// TIA Portal V16 export
// export: Created 2021-07-12T14:47:19.1052506Z, ExportSetting WithDefaults, DisplayName Totally Integrated Automation Portal, DisplayVersion V16, DisplayName TIA Portal Version Control Interface, DisplayVersion V16, DisplayName TIA Portal Openness, DisplayVersion V16, DisplayName STEP 7 Professional, DisplayVersion V16, DisplayName STEP 7 Safety, DisplayVersion V16, DisplayName WinCC Professional, DisplayVersion V16
TYPE "LSimaHydTO_typeDynamicLimits"
TITLE = LSimaHydTO_typeDynamicLimits
// Dynamic limits
// stored: IsFailsafeCompliant false
   STRUCT
      MaxVelocity { S7_SetPoint := 'True'} : LReal := 500.0;   // Maximum permissible velocity of the axis
      MaxAcceleration { S7_SetPoint := 'True'} : LReal := 10000.0;   // Maximum permissible acceleration of the axis
      MaxDeceleration { S7_SetPoint := 'True'} : LReal := 10000.0;   // Maximum permissible deceleration of the axis
      MaxJerk { S7_SetPoint := 'True'} : LReal := 200000.0;   // Maximum permissible jerk on the axis/ not used yet
   END_STRUCT;
END_TYPE
